// Mitsubishi GX Works2 project: 연습   PLC: Q02/Q02H

PROGRAM MAIN
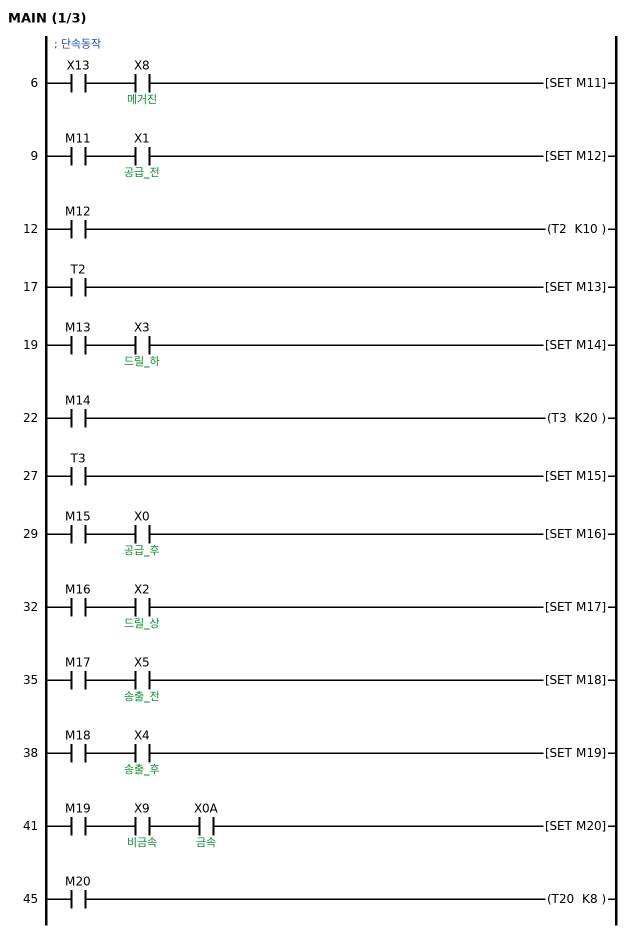
; 단속동작
6     LD      X13
      AND     X8  ; 메거진
      SET     M11
9     LD      M11
      AND     X1  ; 공급_전
      SET     M12
12    LD      M12
      OUT     T2 K10
17    LD      T2
      SET     M13
19    LD      M13
      AND     X3  ; 드릴_하
      SET     M14
22    LD      M14
      OUT     T3 K20
27    LD      T3
      SET     M15
29    LD      M15
      AND     X0  ; 공급_후
      SET     M16
32    LD      M16
      AND     X2  ; 드릴_상
      SET     M17
35    LD      M17
      AND     X5  ; 송출_전
      SET     M18
38    LD      M18
      AND     X4  ; 송출_후
      SET     M19
41    LD      M19
      AND     X9  ; 비금속
      AND     X0A  ; 금속
      SET     M20
45    LD      M20
      OUT     T20 K8
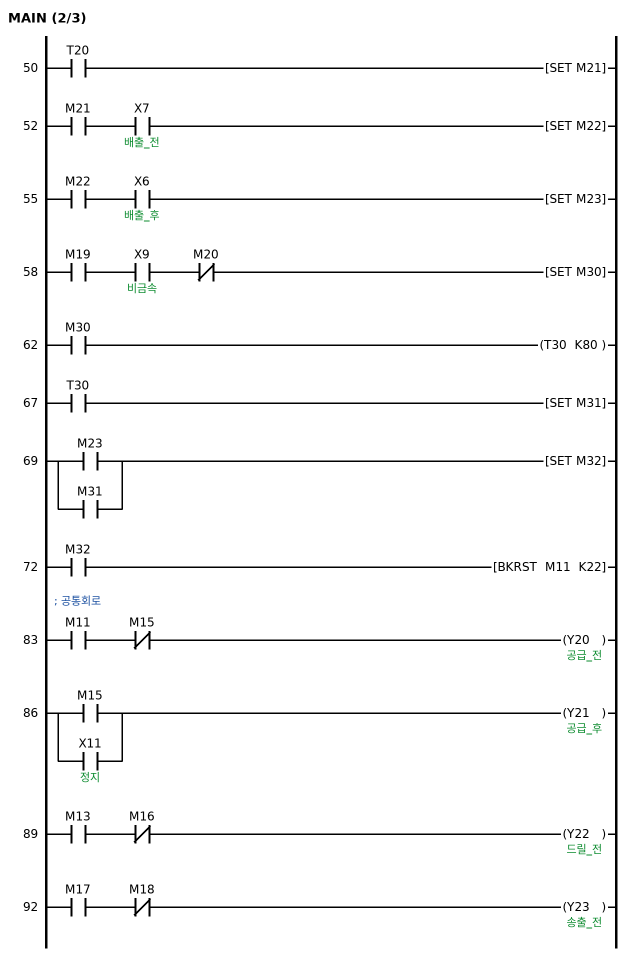
50    LD      T20
      SET     M21
52    LD      M21
      AND     X7  ; 배출_전
      SET     M22
55    LD      M22
      AND     X6  ; 배출_후
      SET     M23
58    LD      M19
      AND     X9  ; 비금속
      ANI     M20
      SET     M30
62    LD      M30
      OUT     T30 K80
67    LD      T30
      SET     M31
69    LD      M23
      OR      M31
      SET     M32
72    LD      M32
      BKRST   M11 K22
; 공통회로
83    LD      M11
      ANI     M15
      OUT     Y20  ; 공급_전
86    LD      M15
      OR      X11  ; 정지
      OUT     Y21  ; 공급_후
89    LD      M13
      ANI     M16
      OUT     Y22  ; 드릴_전
92    LD      M17
      ANI     M18
      OUT     Y23  ; 송출_전
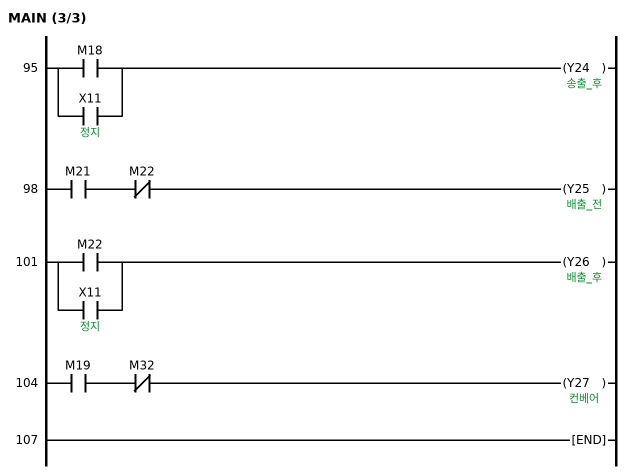
95    LD      M18
      OR      X11  ; 정지
      OUT     Y24  ; 송출_후
98    LD      M21
      ANI     M22
      OUT     Y25  ; 배출_전
101   LD      M22
      OR      X11  ; 정지
      OUT     Y26  ; 배출_후
104   LD      M19
      ANI     M32
      OUT     Y27  ; 컨베어
107   END
END_PROGRAM

// device comments not shown above
X10  ; 시작
Y28  ; 가공드
Y29  ; 적색
Y2A  ; 황색
Y2B  ; 녹색
